{attribute 'GeneratedUsingTerminal: EPP2038-0001-0016'}
{attribute addProperty BoxType "EPP2038-0001-0016"}
{attribute addProperty Id "InputAT %I*BOOL1"}
{attribute addProperty CRC "2198356929"}
{attribute addProperty Size "1"}
TYPE Diag_Channel_830843C1 EXTENDS InputBase_8311D824 :
STRUCT
	{attribute addProperty Name "Input"}
	Input AT %I* : BOOL;
END_STRUCT
END_TYPE

(* stored: Version 1.2.0.0, ProductVersion 3.1.4024.9
   DUT Diag_Channel_830843C1: Id {8b4c8457-bc4c-4c97-b096-dfb2b3d7c01c} *)
